TYPE ST_PNOutput_InputField :
STRUCT
	w_Status					:	WORD;
	w_Warnings					:	WORD;
	w_Faults					:	WORD;
	
	i_ActivePower				:	INT;
	i_ReactivePower				:	INT;
	ui_Frequency				:	UINT;
	ui_VoltageL1N				:	UINT;
	ui_VoltageL2N				:	UINT;
	ui_VoltageL3N				:	UINT;
	ui_VoltageL1L2				:	UINT;
	ui_VoltageL2L3				:	UINT;
	ui_VoltageL3L1				:	UINT;
	i_CurrentL1					:	INT;
	i_CurrentL2					:	INT;
	i_CurrentL3					:	INT;
	i_CurrentN					:	INT;
	ui_TotalEnergySupplied_high :	UINT;
	ui_TotalEnergySupplied_low 	:	UINT;
	ui_TotalEnergyConsumed_high :	UINT;
	ui_TotalEnergyConsumed_low	:	UINT;
END_STRUCT
END_TYPE

(* stored: Version 1.1.0.1, ProductVersion 3.1.4024.12
   DUT ST_PNOutput_InputField: Id {bbea99ac-2297-4afe-bab4-c86f0414e847} *)
